// LS Electric XG5000 project: 런닝머신
// PLC LSPLC

PROGRAM NewProgram (task: 스캔 프로그램)

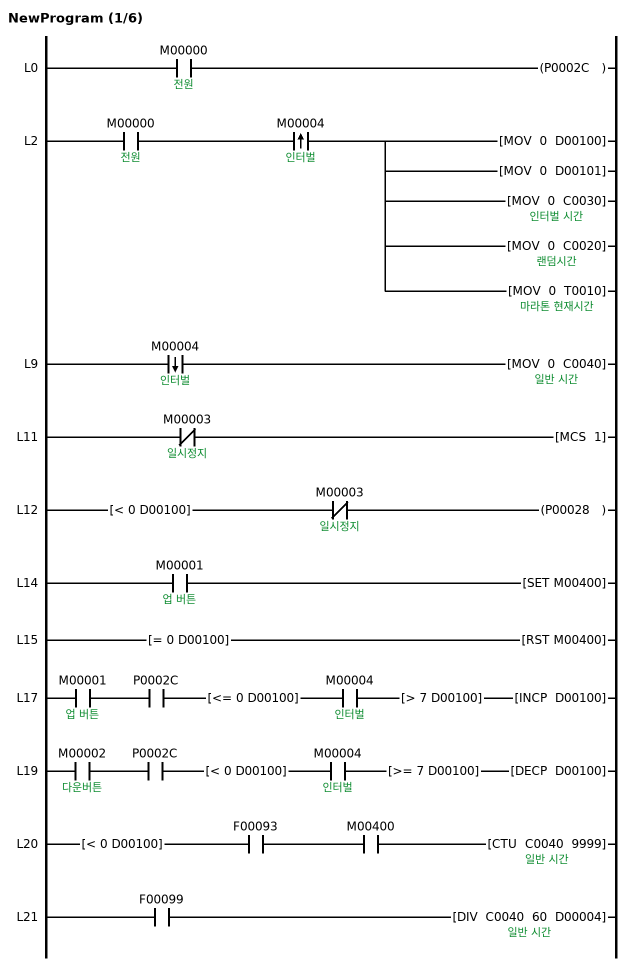
; L0
LOAD      M00000	// 전원
OUT       P0002C
; L2
LOAD      M00000	// 전원
ANDP      M00004	// 인터벌
MOV       0 D00100
MOV       0 D00101
MOV       0 C0030	// 인터벌 시간
MOV       0 C0020	// 랜덤시간
MOV       0 T0010	// 마라톤 현재시간
; L9
LOADN     M00004	// 인터벌
MOV       0 C0040	// 일반 시간
; L11
LOAD NOT  M00003	// 일시정지
MCS       1
; L12
LOAD<     0 D00100
AND NOT   M00003	// 일시정지
OUT       P00028
; L14
LOAD      M00001	// 업 버튼
SET       M00400
; L15
LOAD=     0 D00100
RST       M00400
; L17
LOAD      M00001	// 업 버튼
AND       P0002C
AND<=     0 D00100
AND       M00004	// 인터벌
AND>      7 D00100
INCP      D00100
; L19
LOAD      M00002	// 다운버튼
AND       P0002C
AND<      0 D00100
AND       M00004	// 인터벌
AND>=     7 D00100
DECP      D00100
; L20
LOAD<     0 D00100
AND       F00093
AND       M00400
CTU       C0040 9999	// 일반 시간
; L21
LOAD      F00099
DIV       C0040 60 D00004	// 일반 시간

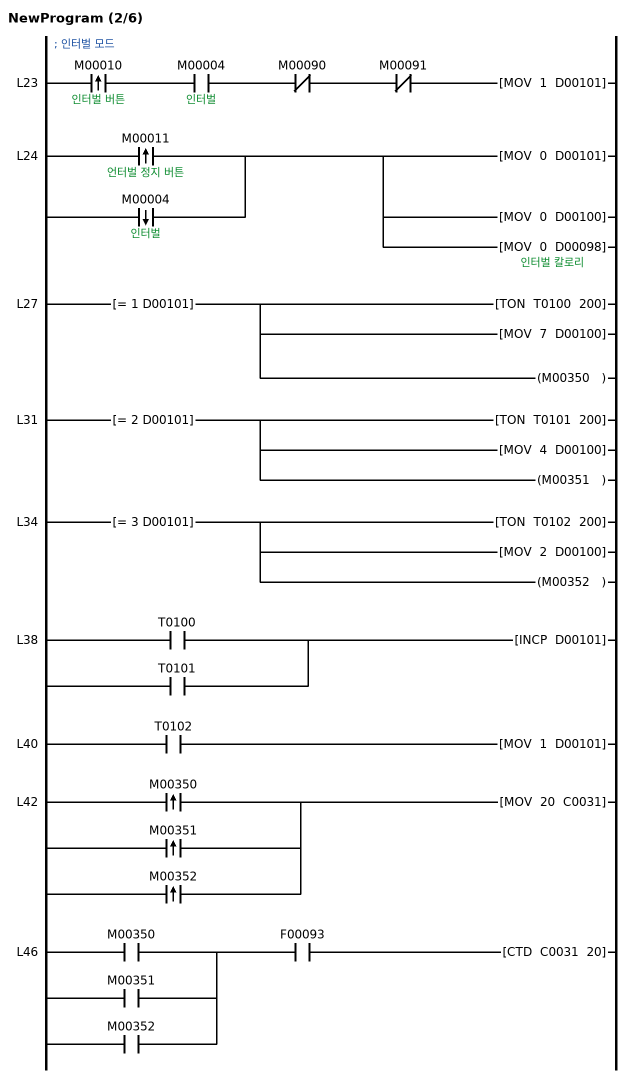
// 인터벌 모드
; L23
LOADP     M00010	// 인터벌 버튼
AND       M00004	// 인터벌
AND NOT   M00090
AND NOT   M00091
MOV       1 D00101
; L24
LOADP     M00011	// 언터벌 정지 버튼
ORN       M00004	// 인터벌
MOV       0 D00101
MOV       0 D00100
MOV       0 D00098	// 인터벌 칼로리
; L27
LOAD=     1 D00101
TON       T0100 200
MOV       7 D00100
OUT       M00350
; L31
LOAD=     2 D00101
TON       T0101 200
MOV       4 D00100
OUT       M00351
; L34
LOAD=     3 D00101
TON       T0102 200
MOV       2 D00100
OUT       M00352
; L38
LOAD      T0100
OR        T0101
INCP      D00101
; L40
LOAD      T0102
MOV       1 D00101
; L42
LOADP     M00350
ORP       M00351
ORP       M00352
MOV       20 C0031
; L46
LOAD      M00350
OR        M00351
OR        M00352
AND       F00093
CTD       C0031 20

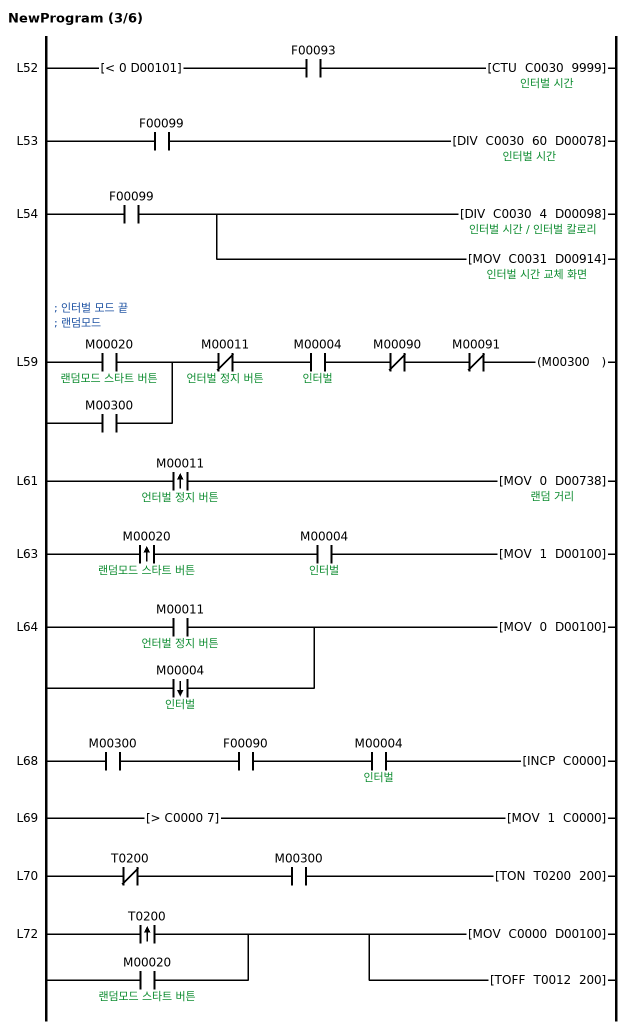
; L52
LOAD<     0 D00101
AND       F00093
CTU       C0030 9999	// 인터벌 시간
; L53
LOAD      F00099
DIV       C0030 60 D00078	// 인터벌 시간
; L54
LOAD      F00099
DIV       C0030 4 D00098	// 인터벌 시간 / 인터벌 칼로리
MOV       C0031 D00914	// 인터벌 시간 교체 화면
// 인터벌 모드 끝
// 랜덤모드
; L59
LOAD      M00020	// 랜덤모드 스타트 버튼
OR        M00300
AND NOT   M00011	// 언터벌 정지 버튼
AND       M00004	// 인터벌
AND NOT   M00090
AND NOT   M00091
OUT       M00300
; L61
LOADP     M00011	// 언터벌 정지 버튼
MOV       0 D00738	// 랜덤 거리
; L63
LOADP     M00020	// 랜덤모드 스타트 버튼
AND       M00004	// 인터벌
MOV       1 D00100
; L64
LOAD      M00011	// 언터벌 정지 버튼
ORN       M00004	// 인터벌
MOV       0 D00100
; L68
LOAD      M00300
AND       F00090
AND       M00004	// 인터벌
INCP      C0000
; L69
LOAD>     C0000 7
MOV       1 C0000
; L70
LOAD NOT  T0200
AND       M00300
TON       T0200 200
; L72
LOADP     T0200
OR        M00020	// 랜덤모드 스타트 버튼
MOV       C0000 D00100
TOFF      T0012 200

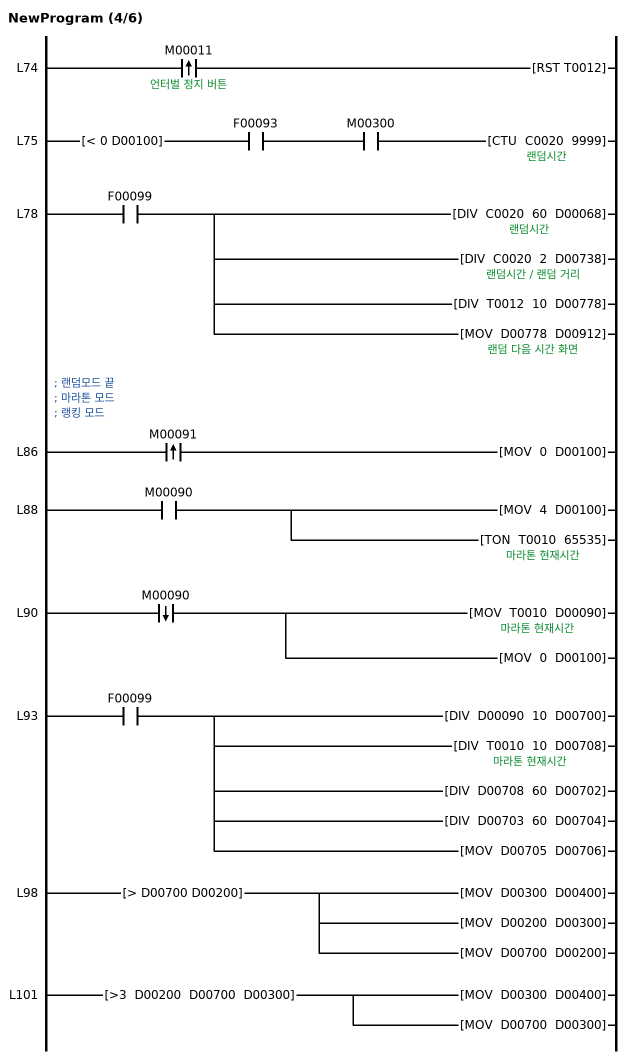
; L74
LOADP     M00011	// 언터벌 정지 버튼
RST       T0012
; L75
LOAD<     0 D00100
AND       F00093
AND       M00300
CTU       C0020 9999	// 랜덤시간
; L78
LOAD      F00099
DIV       C0020 60 D00068	// 랜덤시간
DIV       C0020 2 D00738	// 랜덤시간 / 랜덤 거리
DIV       T0012 10 D00778
MOV       D00778 D00912	// 랜덤 다음 시간 화면
// 랜덤모드 끝
// 마라톤 모드
// 랭킹 모드
; L86
LOADP     M00091
MOV       0 D00100
; L88
LOAD      M00090
MOV       4 D00100
TON       T0010 65535	// 마라톤 현재시간
; L90
LOADN     M00090
MOV       T0010 D00090	// 마라톤 현재시간
MOV       0 D00100
; L93
LOAD      F00099
DIV       D00090 10 D00700
DIV       T0010 10 D00708	// 마라톤 현재시간
DIV       D00708 60 D00702
DIV       D00703 60 D00704
MOV       D00705 D00706
; L98
LOAD>     D00700 D00200
MOV       D00300 D00400
MOV       D00200 D00300
MOV       D00700 D00200
; L101
LOAD>3    D00200 D00700 D00300
MOV       D00300 D00400
MOV       D00700 D00300

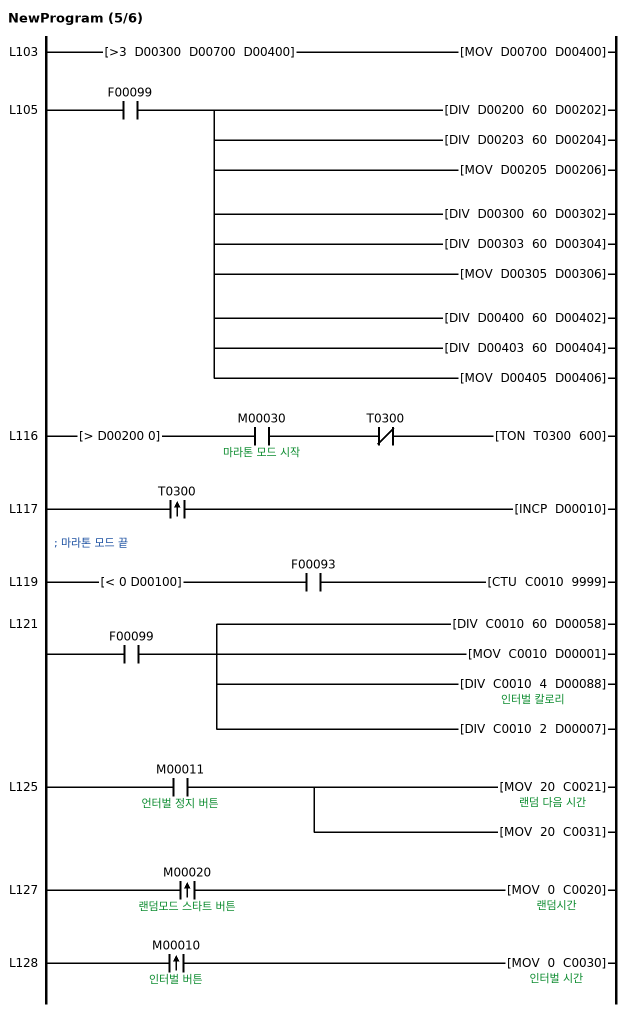
; L103
LOAD>3    D00300 D00700 D00400
MOV       D00700 D00400
; L105
LOAD      F00099
DIV       D00200 60 D00202
DIV       D00203 60 D00204
MOV       D00205 D00206
DIV       D00300 60 D00302
DIV       D00303 60 D00304
MOV       D00305 D00306
DIV       D00400 60 D00402
DIV       D00403 60 D00404
MOV       D00405 D00406
; L116
LOAD>     D00200 0
AND       M00030	// 마라톤 모드 시작
AND NOT   T0300
TON       T0300 600
; L117
LOADP     T0300
INCP      D00010
// 마라톤 모드 끝
; L119
LOAD<     0 D00100
AND       F00093
CTU       C0010 9999
; L121
LOAD      F00099
DIV       C0010 60 D00058
MOV       C0010 D00001
DIV       C0010 4 D00088	// 인터벌 칼로리
DIV       C0010 2 D00007
; L125
LOAD      M00011	// 언터벌 정지 버튼
MOV       20 C0021	// 랜덤 다음 시간
MOV       20 C0031
; L127
LOADP     M00020	// 랜덤모드 스타트 버튼
MOV       0 C0020	// 랜덤시간
; L128
LOADP     M00010	// 인터벌 버튼
MOV       0 C0030	// 인터벌 시간

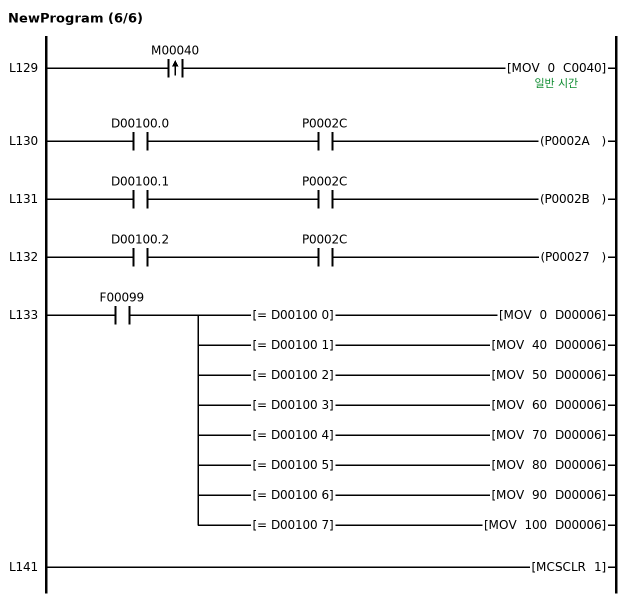
; L129
LOADP     M00040
MOV       0 C0040	// 일반 시간
; L130
LOAD      D00100.0
AND       P0002C
OUT       P0002A
; L131
LOAD      D00100.1
AND       P0002C
OUT       P0002B
; L132
LOAD      D00100.2
AND       P0002C
OUT       P00027
; L133
LOAD      F00099
MPUSH
AND=      D00100 0
MOV       0 D00006
MLOAD
AND=      D00100 1
MOV       40 D00006
MLOAD
AND=      D00100 2
MOV       50 D00006
MLOAD
AND=      D00100 3
MOV       60 D00006
MLOAD
AND=      D00100 4
MOV       70 D00006
MLOAD
AND=      D00100 5
MOV       80 D00006
MLOAD
AND=      D00100 6
MOV       90 D00006
MPOP
AND=      D00100 7
MOV       100 D00006
; L141
MCSCLR    1

VARIABLES AND COMMENTS (devices not used above)
M00100	BIT	인 // 인터벌 작동 릴레이
M00021	BIT	랜덤모드 정지
D00060	WORD	인터벌 설정시간